(* PLC project CODESYS_FourTankProject.project, CODESYS CODESYS V3.5 SP16 *)
(* stored: creationDateTime 2020-05-25T13:01:27.8596011, modificationDateTime 2020-05-25T12:56:40.5524786 *)

PROGRAM PLC_PRG
  VAR
    level1 : REAL;
    pump1 : BOOL;
    valve1 : BOOL;
    full1 : BOOL;
    rate1 : INT;
    vrate1 : INT;
    level2 : REAL;
    pump2 : BOOL;
    valve2 : BOOL;
    full2 : BOOL;
    rate2 : INT;
    vrate2 : INT;
    level3 : REAL;
    pump3 : BOOL;
    valve3 : BOOL;
    full3 : BOOL;
    rate3 : INT;
    vrate3 : INT;
    level4 : REAL;
    pump4 : BOOL;
    valve4 : BOOL;
    full4 : BOOL;
    rate4 : INT;
    vrate4 : INT;
    level0 : REAL;
    pump0 : BOOL;
    valve0 : BOOL;
    full0 : BOOL;
    rate0 : INT;
    vrate0 : INT;
  END_VAR

                    IF level1<100 THEN
	full1:=FALSE; level1:=level1+0.1*rate1/100;
END_IF
IF level1>=0 THEN
	level1:=level1-0.1*vrate1/100;
END_IF
IF level1>=100 THEN
	level1:=100; full1:=TRUE;
END_IF

IF level2<100 THEN
	full2:=FALSE; level2:=level2+0.1*rate2/100;
END_IF
IF level2>=0 THEN
	level2:=level2-0.1*vrate2/100;
END_IF
IF level2>=100 THEN
	level2:=100; full2:=TRUE;
END_IF

IF level3<100 THEN
	full3:=FALSE; level3:=level3+0.1*rate3/100;
END_IF
IF level3>=0 THEN
	level3:=level3-0.1*vrate3/100*1;  
END_IF
IF level3>=100 THEN
	level3:=100; full3:=TRUE;
END_IF

IF level4<100 THEN
	full4:=FALSE; level4:=level4+0.1*rate4/100;
END_IF
IF level4>=0 THEN
	level4:=level4-0.1*vrate4/100;
END_IF
IF level4>=100 THEN
	level4:=100; full4:=TRUE;
END_IF

level0:=100-(level1+level2+level3+level4)/4;
IF rate1>0 AND (level0>0 OR (valve1 OR valve2 OR valve3 OR valve4)) THEN pump1:=TRUE; ELSE pump1:=FALSE; END_IF
IF rate2>0 AND (level0>0 OR (valve1 OR valve2 OR valve3 OR valve4)) THEN pump2:=TRUE; ELSE pump2:=FALSE; END_IF
IF rate3>0 AND (level0>0 OR (valve1 OR valve2 OR valve3 OR valve4)) THEN pump3:=TRUE; ELSE pump3:=FALSE; END_IF
IF rate4>0 AND (level0>0 OR (valve1 OR valve2 OR valve3 OR valve4)) THEN pump4:=TRUE; ELSE pump4:=FALSE; END_IF

IF vrate1>0 AND (level1>0 OR pump1=TRUE) THEN valve1:=TRUE; ELSE valve1:=FALSE; END_IF
IF vrate2>0 AND (level2>0 OR pump2=TRUE) THEN valve2:=TRUE; ELSE valve2:=FALSE; END_IF
IF vrate3>0 AND (level3>0 OR pump3=TRUE) THEN valve3:=TRUE; ELSE valve3:=FALSE; END_IF
IF vrate4>0 AND (level4>0 OR pump4=TRUE) THEN valve4:=TRUE; ELSE valve4:=FALSE; END_IF
	
IF level0=0 THEN full1:=FALSE; full2:=FALSE; full3:=FALSE; full4:=FALSE; END_IF

                  
END_PROGRAM

CONFIGURATION Device
  RESOURCE Application ON PLC
    TASK MainTask(INTERVAL := T#10ms, PRIORITY := 1);
    TASK VISU_TASK(INTERVAL := T#100ms, PRIORITY := 31);
    PROGRAM PLC_PRG WITH MainTask : PLC_PRG;
    PROGRAM VisuElems.Visu_Prg WITH VISU_TASK : VisuElems.Visu_Prg;
  END_RESOURCE
END_CONFIGURATION
